FUNCTION_BLOCK FB_PM_Base 
//////////////////
// Measurement Solution. Base FB
//////////////////
VAR_INPUT PERSISTENT
	// Parameters of the Object (instance specific) 
	ParamTempoComAlarm				: TIME 		:= T#10S ; 						(* (s) Config : Tempo to detect LOC Alarm*)
	{attribute 'OPC.UA.DA' := '1'} 
	ParamClockReadTime 				: TIME 		:= TIME#200MS;	  				(* (ms) Read Modbus period  *)
	ParamTimeout					: TIME  	:= T#2S ;			  			(* (s) Timeout for modbus reading*)
	
	
END_VAR

VAR_INPUT
	//Child objects
	IN_CmdToggleRead				: BOOL ; 
	IN_CmdReset_L					: BOOL ;									// (NA) External Reset Command

END_VAR
VAR
	//M_ALARMMANAGEMENT VARIABLES//
		TON_ComAlarm				: TON ; 									// Tempo before detecting loss of communication 
	    TON_ComWarning				: TON ; 									// Tempo before detecting loss of one frame                                               								
                                            								    
		MesWarningCom				: BOOL ; 									// True if bad communication 
                                                                                 
	//M_READ VARIABLES//                                                         
//	MesDataExd		AT %Q*	: PM ;                                 
		ClockRead			AT %Q*	: BOOL ;	 								// Clock Read
                                                                                
		                                                                         
	//M_INIT VARIABLES //
		bInit						: BOOL 				:= TRUE ; 							// (NA) Initialize object parameters at first cycle 
		                                                                         
	// M_EXECUTE VARIABLES //
		TP1							: TP ; 												// (NA) Tempo to define Modbus Reading Frequency  
                                                             	                                                                                                                                                      
		//MesCP_Read					: BOOL;													// (NA) Permanent conditions to activate method
        Trig_Cmd_Read				: R_TRIG;      

                 
END_VAR

METHOD M_AlarmManagement
//////////////////
// Digiware measurement tool alarm and warning management
/////////////////

VAR 
	
END_VAR
END_METHOD

METHOD M_CP
//////////////////
//  Emulator
/////////////////

VAR 
	// Method local variables (reinitialized at each cycle) 
	
END_VAR
END_METHOD

METHOD M_Execute
//////////////////
//  Method Calls 
/////////////////
VAR 
	// Method local variables (reinitialized at each cycle) 
	// EMULATOR

	
END_VAR
// READING AND WRITING CLOCK //
	TP1(IN:=NOT TP1.Q , PT:= ParamClockReadTime);
	ClockRead 		:= TP1.Q;

// PERMANENT CONDITIONS //
	M_CP() ; 
	
// METHODS CALLS //
	IF bInit THEN
		M_Init() ; 
		bInit					:= FALSE ; 
	ELSIF CmdInit_G OR IN_CmdReset_L THEN 
		bInit:= TRUE ;		
	END_IF

	M_Read() ; 
	M_AlarmManagement();
END_METHOD

METHOD M_Init
VAR 

END_VAR
END_METHOD

METHOD M_Read
//////////////////
//  Read Modbus Variable for PCS . 
/////////////////
VAR 
	// Method local variables (reinitialized at each cycle) 
	
END_VAR
END_METHOD

END_FUNCTION_BLOCK

(* stored: Version 1.1.0.1
   POU FB_PM_Base: Id {d03ca925-83b8-453a-a2ed-fabfea0c87ea}, SpecialFunc None
   Method M_AlarmManagement: Id {55f37f90-d101-4087-ae83-23902e38e74d}
   Method M_CP: Id {b84f0547-cdae-4a37-ad2e-c36249718d09}
   Method M_Execute: Id {69ed72c7-fa2c-4bbc-ad69-38d92c70dd44}
   Method M_Init: Id {509d3645-b00a-4fd8-aae1-e1d2fae3b32d}
   Method M_Read: Id {56465a00-ea0b-4f7d-89af-61c6317771ac} *)
